// TIA Portal V19 export
DATA_BLOCK "A02_Config"   // DB38
// stored: MemoryReserve 100
   VAR RETAIN
      Area02_Main { ExternalAccessible := 'False'; ExternalVisible := 'False'; ExternalWritable := 'False'} : "AreaConfig";
      RollformingMng : Struct
         SensorsDelayOn : Time := T#100MS;
         SensorsDelayOff : Time := T#500MS;
         SensorExtractor_DelayOn : Time := T#250MS;
         SensorExtractor_DelayOff : Time := T#100MS;
      END_STRUCT;
      PitTableLoop1 : Struct
         LIFT : "ValveMachine_Config";
         Exist : Bool := TRUE;
      END_STRUCT;
      A0201_Profilatrice_RegolazioneFormato : Struct
         Ax_D : Array[1..6] of "Positioning_DOL_Machine_Config";
         Ax_M : Array[7..14] of "Positioning_MOL_Machine_Config";
      END_STRUCT;
      Area02_HU { ExternalAccessible := 'False'; ExternalVisible := 'False'; ExternalWritable := 'False'} : Struct
         Pump { S7_SetPoint := 'True'} : "HU_Pump_Config";
         Tank { S7_SetPoint := 'True'} : "HU_Tank_Config";
      END_STRUCT;
      PostPunchingMatCounter : Struct
         Default_FAK : LReal := 1.0;
      END_STRUCT;
      Rollformer : "PositioningMachine_Config";
      RollfomerLubr { S7_SetPoint := 'True'} : "LubrValve_Config";
      MwFakCalc : Struct
         PushAx : "SpeedMachine_Config";
         Gripper : "ValveMachine_Config";
         MaterialPresenceDly : Time := T#250MS;
         MaterialAbsenceDly : Time := T#250MS;
         PushAx_FwdTimeout { ExternalAccessible := 'False'; ExternalVisible := 'False'; ExternalWritable := 'False'} : Time := T#30S;
         PushAx_BwdTimeout { ExternalAccessible := 'False'; ExternalVisible := 'False'; ExternalWritable := 'False'} : Time := T#30S;
         Default_FAK : LReal := 1.0;
      END_STRUCT;
      FlyingCarriage : "udt_FlyingCarriage_Config";
      FinalCut : Struct
         CheckRestPosition : Bool := TRUE;
         CutHead : "ValveMachine_Config";
         DrawHead : "ValveMachine_Config";
         MarkHead : "ValveMachine_Config";
         Locking : "ValveMachine_Config";
         Locking_AI_HighLimit : Real := 250.0;
         Locking_AI_LowLimit : Real := 0.0;
      END_STRUCT;
      FinalCutLub : Struct
         EnableWngSystemOff : Bool := FALSE;
         ExternalPump : Bool := FALSE;
         PumpWorkDuration : Time := T#2S;
         PumpPauseDuration : Time := T#3S;
         LowTankLevelDly : Time := T#3S;
      END_STRUCT;
      AccRollConveyor : Struct
         Roll1 : "SpeedMachine_Config";
         Roll2 : "SpeedMachine_Config";
         Roll3 : "SpeedMachine_Config";
         PusherVert : Array[1..6] of "ValveMachine_Config";
         PusherHoriz : Array[1..6] of "ValveMachine_Config";
         SensorsDelayOn : Time := T#10MS;
         SensorsDelayOff : Time := T#10MS;
         ExitLeftDelayOn : Time := T#250MS;
         ExitLeftDelayOff : Time := T#250MS;
      END_STRUCT;
   END_VAR
BEGIN
   Area02_Main.TimeOutStopImmediate := T#2S;
   Area02_Main.TimeOutStopInPhase := T#30S;
   Area02_Main.TimeOutStopProgrammed := T#1M;
   Area02_Main.TimeOutResetAlarms := T#1S;
   PitTableLoop1.LIFT.DelayPressureRunningTimeout := T#3S;
   PitTableLoop1.LIFT.DelayMissingCondition := T#3S;
   PitTableLoop1.LIFT.Rest_LsQty := 1;
   PitTableLoop1.LIFT.Work_LsQty := 1;
   PitTableLoop1.LIFT.Rest_RetainAut := FALSE;
   PitTableLoop1.LIFT.Work_RetainAut := FALSE;
   PitTableLoop1.LIFT.V.RestLimSwitchExist := TRUE;
   PitTableLoop1.LIFT.V.WorkLimSwitchExist := TRUE;
   PitTableLoop1.LIFT.V.CheckOilInPressure := FALSE;
   PitTableLoop1.LIFT.V.CutRestWhenIsAtRest := FALSE;
   PitTableLoop1.LIFT.V.CutWorkWhenIsAtWork := FALSE;
   PitTableLoop1.LIFT.V.RestTime := T#1MS;
   PitTableLoop1.LIFT.V.WorkTime := T#1MS;
   PitTableLoop1.LIFT.V.RestTimeOut := T#10S;
   PitTableLoop1.LIFT.V.WorkTimeOut := T#10S;
   A0201_Profilatrice_RegolazioneFormato.Ax_D[1..6].DelayMissingCondition := T#3S;
   A0201_Profilatrice_RegolazioneFormato.Ax_D[1..6].CyclicOBTime_ms := 10.0;
   A0201_Profilatrice_RegolazioneFormato.Ax_D[1..6].Ax.limitMinus := 0.0;
   A0201_Profilatrice_RegolazioneFormato.Ax_D[1..6].Ax.limitPlus := 0.0;
   A0201_Profilatrice_RegolazioneFormato.Ax_D[1..6].Ax.Backlash := 0.4;
   A0201_Profilatrice_RegolazioneFormato.Ax_D[1..6].Ax.BacklashActivation := TRUE;
   A0201_Profilatrice_RegolazioneFormato.Ax_D[1..6].Ax.ToleranceWindow := 0.0;
   A0201_Profilatrice_RegolazioneFormato.Ax_D[1..6].Ax.ToleranceWindowDelay := T#100MS;
   A0201_Profilatrice_RegolazioneFormato.Ax_D[1..6].Ax.PreCutOff := 0.0;
   A0201_Profilatrice_RegolazioneFormato.Ax_D[1..6].Ax.PreEndLowSpeed := 0.0;
   A0201_Profilatrice_RegolazioneFormato.Ax_D[1..6].Ax.PreEndMedSpeed := 0.0;
   A0201_Profilatrice_RegolazioneFormato.Ax_D[1..6].Ax.ChangeDirectionDelay := T#0MS;
   A0201_Profilatrice_RegolazioneFormato.Ax_D[1..6].Ax.StandstillVelocity := 0.5;
   A0201_Profilatrice_RegolazioneFormato.Ax_D[1..6].Ax.StandStillDelay := T#100MS;
   A0201_Profilatrice_RegolazioneFormato.Ax_D[1..6].Ax.HomingDirection := FALSE;
   A0201_Profilatrice_RegolazioneFormato.Ax_D[1..6].Ax.RecallTime := 0.0;
   A0201_Profilatrice_RegolazioneFormato.Ax_D[1..6].Ax.VelocityFilter_T := 10.0;
   A0201_Profilatrice_RegolazioneFormato.Ax_D[1..6].Ax.VelocityMeasUnit := 2;
   A0201_Profilatrice_RegolazioneFormato.Ax_D[1..6].Ax.PosFbkDisabled := FALSE;
   A0201_Profilatrice_RegolazioneFormato.Ax_D[1..6].Ax.FbkCtrlDisabled := TRUE;
   A0201_Profilatrice_RegolazioneFormato.Ax_D[1..6].Ax_UM2."m" := -1.0;
   A0201_Profilatrice_RegolazioneFormato.Ax_D[1].Ax_UM2.q := 267.4;
   A0201_Profilatrice_RegolazioneFormato.Ax_D[2].Ax_UM2.q := 267.3;
   A0201_Profilatrice_RegolazioneFormato.Ax_D[3].Ax_UM2.q := 262.3;
   A0201_Profilatrice_RegolazioneFormato.Ax_D[4].Ax_UM2.q := 262.6;
   A0201_Profilatrice_RegolazioneFormato.Ax_D[5].Ax_UM2.q := 261.8;
   A0201_Profilatrice_RegolazioneFormato.Ax_D[6].Ax_UM2.q := 262.0;
   A0201_Profilatrice_RegolazioneFormato.Ax_D[1..6].S120.SpeedMotor.ReferenceVelocity := 2200.0;
   A0201_Profilatrice_RegolazioneFormato.Ax_D[1..6].S120.SpeedMotor.InvertDirection := FALSE;
   A0201_Profilatrice_RegolazioneFormato.Ax_D[1..6].S120.PowerOffDelay := T#1S_500MS;
   A0201_Profilatrice_RegolazioneFormato.Ax_D[1..6].S120.StandstillVelocity := 20.0;
   A0201_Profilatrice_RegolazioneFormato.Ax_D[1..6].S120.AccTime := 0.5;
   A0201_Profilatrice_RegolazioneFormato.Ax_D[1..6].S120.DecTime := 0.5;
   A0201_Profilatrice_RegolazioneFormato.Ax_D[1..6].Fan.Presence := FALSE;
   A0201_Profilatrice_RegolazioneFormato.Ax_D[1..6].Fan.DelayOff := T#10M;
   A0201_Profilatrice_RegolazioneFormato.Ax_D[1..6].Brake_Presence := FALSE;
   A0201_Profilatrice_RegolazioneFormato.Ax_M[7..14].DelayMissingCondition := T#0MS;
   A0201_Profilatrice_RegolazioneFormato.Ax_M[7..14].CyclicOBTime_ms := 10.0;
   A0201_Profilatrice_RegolazioneFormato.Ax_M[7..14].Ax.limitMinus := 0.0;
   A0201_Profilatrice_RegolazioneFormato.Ax_M[7..14].Ax.limitPlus := 0.0;
   A0201_Profilatrice_RegolazioneFormato.Ax_M[7..14].Ax.Backlash := 0.4;
   A0201_Profilatrice_RegolazioneFormato.Ax_M[7..14].Ax.BacklashActivation := TRUE;
   A0201_Profilatrice_RegolazioneFormato.Ax_M[7..14].Ax.ToleranceWindow := 0.0;
   A0201_Profilatrice_RegolazioneFormato.Ax_M[7..14].Ax.ToleranceWindowDelay := T#100MS;
   A0201_Profilatrice_RegolazioneFormato.Ax_M[7..14].Ax.PreCutOff := 0.0;
   A0201_Profilatrice_RegolazioneFormato.Ax_M[7..14].Ax.PreEndLowSpeed := 0.0;
   A0201_Profilatrice_RegolazioneFormato.Ax_M[7..14].Ax.PreEndMedSpeed := 0.0;
   A0201_Profilatrice_RegolazioneFormato.Ax_M[7..14].Ax.ChangeDirectionDelay := T#0MS;
   A0201_Profilatrice_RegolazioneFormato.Ax_M[7..14].Ax.StandstillVelocity := 0.5;
   A0201_Profilatrice_RegolazioneFormato.Ax_M[7..14].Ax.StandStillDelay := T#100MS;
   A0201_Profilatrice_RegolazioneFormato.Ax_M[7..14].Ax.HomingDirection := FALSE;
   A0201_Profilatrice_RegolazioneFormato.Ax_M[7..14].Ax.RecallTime := 0.0;
   A0201_Profilatrice_RegolazioneFormato.Ax_M[7..14].Ax.VelocityFilter_T := 10.0;
   A0201_Profilatrice_RegolazioneFormato.Ax_M[7..14].Ax.VelocityMeasUnit := 2;
   A0201_Profilatrice_RegolazioneFormato.Ax_M[7..14].Ax.PosFbkDisabled := FALSE;
   A0201_Profilatrice_RegolazioneFormato.Ax_M[7..14].Ax.FbkCtrlDisabled := TRUE;
   A0201_Profilatrice_RegolazioneFormato.Ax_M[7..8].Ax_UM2."m" := -1.0;
   A0201_Profilatrice_RegolazioneFormato.Ax_M[9..10].Ax_UM2."m" := 1.0;
   A0201_Profilatrice_RegolazioneFormato.Ax_M[11..14].Ax_UM2."m" := -1.0;
   A0201_Profilatrice_RegolazioneFormato.Ax_M[7..8].Ax_UM2.q := 84.8;
   A0201_Profilatrice_RegolazioneFormato.Ax_M[9..10].Ax_UM2.q := 0.0;
   A0201_Profilatrice_RegolazioneFormato.Ax_M[11..12].Ax_UM2.q := 81.6;
   A0201_Profilatrice_RegolazioneFormato.Ax_M[13..14].Ax_UM2.q := 81.3;
   Area02_HU.Pump.SafetyCutOffValveExist := TRUE;
   Area02_HU.Pump.StandbyValveExist := TRUE;
   Area02_HU.Pump.OilPumpContactotFeedbackTimeOut := T#5S;
   Area02_HU.Tank.RecirculationPumpExist := TRUE;
   Area02_HU.Tank.HeatExchangerFanExist := TRUE;
   Area02_HU.Tank.HeatingUnitExistNum := 1;
   Area02_HU.Tank.ChillerExist := FALSE;
   Area02_HU.Tank.OilMaxTemperature := 70.0;
   Area02_HU.Tank.WaterMaxTemperature := 60.0;
   Area02_HU.Tank.TemperatureStartCheckFilters := 35.0;
   Area02_HU.Tank.HeatingHysteresys := 1.0;
   Area02_HU.Tank.DelayHeatingStart := T#30S;
   Area02_HU.Tank.DelayHeatingStop := T#30S;
   Area02_HU.Tank.DelayCollingStart := T#30S;
   Area02_HU.Tank.DelayCollingStop := T#30S;
   Area02_HU.Tank.AnlOilTemp_HighLimit := 100.0;
   Area02_HU.Tank.AnlOilTemp_LowLimit := 0.0;
   Area02_HU.Tank.AnlWaterTemp_HighLimit := 100.0;
   Area02_HU.Tank.AnlWaterTemp_LowLimit := -10.0;
   Rollformer.SLS_VEL := 5000.0;
   Rollformer.DelayMissingCondition := T#3S;
   Rollformer.Ax.OptionON_EncoderSelection := FALSE;
   Rollformer.Ax.OptionON_ParameterChange := TRUE;
   Rollformer.Ax.OptionON_AutoReloadPosition := TRUE;
   Rollformer.Ax.OptionON_ManPreset := FALSE;
   Rollformer.Ax.HomeMode := 0;
   Rollformer.Ax.PosAxis.Simulation := FALSE;
   Rollformer.Ax.PosAxis.PowerOffDelay := T#5S;
   Rollformer.Ax.PosAxis.PowerStartMode := 1;
   Rollformer.Ax.PosAxis.PowerStopMode := 2;
   Rollformer.Fan.Presence := TRUE;
   Rollformer.Fan.DelayOff := T#10M;
   Rollformer.Brake_Presence := FALSE;
   RollfomerLubr.WorkMode := 2;
   RollfomerLubr.CounterMode := 0;
   RollfomerLubr.ValveType := 1;
   RollfomerLubr.ManualCmdTimeOut := T#5M;
   MwFakCalc.PushAx.SLS_VEL := 5000.0;
   MwFakCalc.PushAx.DelayMissingCondition := T#3S;
   MwFakCalc.PushAx.Ax.SINA_Drive.ReferenceVelocity := 2200.0;
   MwFakCalc.PushAx.Ax.SINA_Drive.InvertDirection := FALSE;
   MwFakCalc.PushAx.Ax.MinAccTime := 0.1;
   MwFakCalc.PushAx.Ax.MinDecTime := 0.1;
   MwFakCalc.PushAx.Ax.LeadScrewPitchVal := 79.984948;
   MwFakCalc.PushAx.Ax.MotorRevolution := 5.0;
   MwFakCalc.PushAx.Ax.LoadRevolution := 1.0;
   MwFakCalc.PushAx.Ax.PowerOffDelay := T#1S_500MS;
   MwFakCalc.PushAx.Ax.StandstillVelocity := 20.0;
   MwFakCalc.PushAx.Ax.StandstillDelay := T#100MS;
   MwFakCalc.PushAx.Fan.Presence := FALSE;
   MwFakCalc.PushAx.Fan.DelayOff := T#0MS;
   MwFakCalc.PushAx.Brake_Presence := FALSE;
   MwFakCalc.Gripper.DelayPressureRunningTimeout := T#3S;
   MwFakCalc.Gripper.DelayMissingCondition := T#3S;
   MwFakCalc.Gripper.Rest_LsQty := 1;
   MwFakCalc.Gripper.Work_LsQty := 1;
   MwFakCalc.Gripper.Rest_RetainAut := FALSE;
   MwFakCalc.Gripper.Work_RetainAut := FALSE;
   MwFakCalc.Gripper.V.RestLimSwitchExist := TRUE;
   MwFakCalc.Gripper.V.WorkLimSwitchExist := TRUE;
   MwFakCalc.Gripper.V.CheckOilInPressure := FALSE;
   MwFakCalc.Gripper.V.CutRestWhenIsAtRest := TRUE;
   MwFakCalc.Gripper.V.CutWorkWhenIsAtWork := TRUE;
   MwFakCalc.Gripper.V.RestTime := T#1MS;
   MwFakCalc.Gripper.V.WorkTime := T#1MS;
   MwFakCalc.Gripper.V.RestTimeOut := T#1S;
   MwFakCalc.Gripper.V.WorkTimeOut := T#1S;
   FlyingCarriage.SLS_VEL := 5000.0;
   FlyingCarriage.DelayMissingCondition := T#3S;
   FlyingCarriage.Fan.Exist := FALSE;
   FlyingCarriage.Fan.DelayOff := T#15M;
   FinalCut.CutHead.DelayPressureRunningTimeout := T#3S;
   FinalCut.CutHead.DelayMissingCondition := T#3S;
   FinalCut.CutHead.Rest_LsQty := 1;
   FinalCut.CutHead.Work_LsQty := 1;
   FinalCut.CutHead.Rest_RetainAut := FALSE;
   FinalCut.CutHead.Work_RetainAut := FALSE;
   FinalCut.CutHead.V.RestLimSwitchExist := TRUE;
   FinalCut.CutHead.V.WorkLimSwitchExist := TRUE;
   FinalCut.CutHead.V.CheckOilInPressure := TRUE;
   FinalCut.CutHead.V.CutRestWhenIsAtRest := FALSE;
   FinalCut.CutHead.V.CutWorkWhenIsAtWork := FALSE;
   FinalCut.CutHead.V.RestTime := T#1MS;
   FinalCut.CutHead.V.WorkTime := T#1MS;
   FinalCut.CutHead.V.RestTimeOut := T#1S_500MS;
   FinalCut.CutHead.V.WorkTimeOut := T#1S_500MS;
   FinalCut.DrawHead.DelayPressureRunningTimeout := T#3S;
   FinalCut.DrawHead.DelayMissingCondition := T#3S;
   FinalCut.DrawHead.Rest_LsQty := 1;
   FinalCut.DrawHead.Work_LsQty := 1;
   FinalCut.DrawHead.Rest_RetainAut := FALSE;
   FinalCut.DrawHead.Work_RetainAut := FALSE;
   FinalCut.DrawHead.V.RestLimSwitchExist := TRUE;
   FinalCut.DrawHead.V.WorkLimSwitchExist := TRUE;
   FinalCut.DrawHead.V.CheckOilInPressure := TRUE;
   FinalCut.DrawHead.V.CutRestWhenIsAtRest := FALSE;
   FinalCut.DrawHead.V.CutWorkWhenIsAtWork := FALSE;
   FinalCut.DrawHead.V.RestTime := T#1MS;
   FinalCut.DrawHead.V.WorkTime := T#1MS;
   FinalCut.DrawHead.V.RestTimeOut := T#1S_500MS;
   FinalCut.DrawHead.V.WorkTimeOut := T#1S_500MS;
   FinalCut.MarkHead.DelayPressureRunningTimeout := T#3S;
   FinalCut.MarkHead.DelayMissingCondition := T#3S;
   FinalCut.MarkHead.Rest_LsQty := 1;
   FinalCut.MarkHead.Work_LsQty := 1;
   FinalCut.MarkHead.Rest_RetainAut := FALSE;
   FinalCut.MarkHead.Work_RetainAut := FALSE;
   FinalCut.MarkHead.V.RestLimSwitchExist := TRUE;
   FinalCut.MarkHead.V.WorkLimSwitchExist := TRUE;
   FinalCut.MarkHead.V.CheckOilInPressure := TRUE;
   FinalCut.MarkHead.V.CutRestWhenIsAtRest := FALSE;
   FinalCut.MarkHead.V.CutWorkWhenIsAtWork := FALSE;
   FinalCut.MarkHead.V.RestTime := T#1MS;
   FinalCut.MarkHead.V.WorkTime := T#1MS;
   FinalCut.MarkHead.V.RestTimeOut := T#1S_500MS;
   FinalCut.MarkHead.V.WorkTimeOut := T#1S_500MS;
   FinalCut.Locking.DelayPressureRunningTimeout := T#3S;
   FinalCut.Locking.DelayMissingCondition := T#3S;
   FinalCut.Locking.Rest_LsQty := 1;
   FinalCut.Locking.Work_LsQty := 1;
   FinalCut.Locking.Rest_RetainAut := FALSE;
   FinalCut.Locking.Work_RetainAut := FALSE;
   FinalCut.Locking.V.RestLimSwitchExist := TRUE;
   FinalCut.Locking.V.WorkLimSwitchExist := TRUE;
   FinalCut.Locking.V.CheckOilInPressure := TRUE;
   FinalCut.Locking.V.CutRestWhenIsAtRest := FALSE;
   FinalCut.Locking.V.CutWorkWhenIsAtWork := FALSE;
   FinalCut.Locking.V.RestTime := T#1MS;
   FinalCut.Locking.V.WorkTime := T#1MS;
   FinalCut.Locking.V.RestTimeOut := T#2S;
   FinalCut.Locking.V.WorkTimeOut := T#2S;
   AccRollConveyor.Roll1.SLS_VEL := 5000.0;
   AccRollConveyor.Roll1.DelayMissingCondition := T#3S;
   AccRollConveyor.Roll1.Ax.SINA_Drive.ReferenceVelocity := 2200.0;
   AccRollConveyor.Roll1.Ax.SINA_Drive.InvertDirection := FALSE;
   AccRollConveyor.Roll1.Ax.MinAccTime := 0.1;
   AccRollConveyor.Roll1.Ax.MinDecTime := 0.1;
   AccRollConveyor.Roll1.Ax.LeadScrewPitchVal := 219.911;
   AccRollConveyor.Roll1.Ax.MotorRevolution := 7.0;
   AccRollConveyor.Roll1.Ax.LoadRevolution := 1.0;
   AccRollConveyor.Roll1.Ax.PowerOffDelay := T#1S_500MS;
   AccRollConveyor.Roll1.Ax.StandstillVelocity := 50.0;
   AccRollConveyor.Roll1.Ax.StandstillDelay := T#100MS;
   AccRollConveyor.Roll1.Fan.Presence := FALSE;
   AccRollConveyor.Roll1.Fan.DelayOff := T#0MS;
   AccRollConveyor.Roll1.Brake_Presence := FALSE;
   AccRollConveyor.Roll2.SLS_VEL := 5000.0;
   AccRollConveyor.Roll2.DelayMissingCondition := T#3S;
   AccRollConveyor.Roll2.Ax.SINA_Drive.ReferenceVelocity := 2200.0;
   AccRollConveyor.Roll2.Ax.SINA_Drive.InvertDirection := FALSE;
   AccRollConveyor.Roll2.Ax.MinAccTime := 0.1;
   AccRollConveyor.Roll2.Ax.MinDecTime := 0.1;
   AccRollConveyor.Roll2.Ax.LeadScrewPitchVal := 219.911;
   AccRollConveyor.Roll2.Ax.MotorRevolution := 7.0;
   AccRollConveyor.Roll2.Ax.LoadRevolution := 1.0;
   AccRollConveyor.Roll2.Ax.PowerOffDelay := T#1S_500MS;
   AccRollConveyor.Roll2.Ax.StandstillVelocity := 50.0;
   AccRollConveyor.Roll2.Ax.StandstillDelay := T#100MS;
   AccRollConveyor.Roll2.Fan.Presence := FALSE;
   AccRollConveyor.Roll2.Fan.DelayOff := T#0MS;
   AccRollConveyor.Roll2.Brake_Presence := FALSE;
   AccRollConveyor.Roll3.SLS_VEL := 5000.0;
   AccRollConveyor.Roll3.DelayMissingCondition := T#3S;
   AccRollConveyor.Roll3.Ax.SINA_Drive.ReferenceVelocity := 2200.0;
   AccRollConveyor.Roll3.Ax.SINA_Drive.InvertDirection := FALSE;
   AccRollConveyor.Roll3.Ax.MinAccTime := 0.1;
   AccRollConveyor.Roll3.Ax.MinDecTime := 0.1;
   AccRollConveyor.Roll3.Ax.LeadScrewPitchVal := 219.911;
   AccRollConveyor.Roll3.Ax.MotorRevolution := 7.0;
   AccRollConveyor.Roll3.Ax.LoadRevolution := 1.0;
   AccRollConveyor.Roll3.Ax.PowerOffDelay := T#1S_500MS;
   AccRollConveyor.Roll3.Ax.StandstillVelocity := 50.0;
   AccRollConveyor.Roll3.Ax.StandstillDelay := T#100MS;
   AccRollConveyor.Roll3.Fan.Presence := FALSE;
   AccRollConveyor.Roll3.Fan.DelayOff := T#0MS;
   AccRollConveyor.Roll3.Brake_Presence := FALSE;
   AccRollConveyor.PusherVert[1..6].DelayPressureRunningTimeout := T#3S;
   AccRollConveyor.PusherVert[1..6].DelayMissingCondition := T#3S;
   AccRollConveyor.PusherVert[1..6].Rest_LsQty := 1;
   AccRollConveyor.PusherVert[1..6].Work_LsQty := 1;
   AccRollConveyor.PusherVert[1..6].Rest_RetainAut := FALSE;
   AccRollConveyor.PusherVert[1..6].Work_RetainAut := FALSE;
   AccRollConveyor.PusherVert[1..6].V.RestLimSwitchExist := TRUE;
   AccRollConveyor.PusherVert[1..6].V.WorkLimSwitchExist := FALSE;
   AccRollConveyor.PusherVert[1..6].V.CheckOilInPressure := FALSE;
   AccRollConveyor.PusherVert[1..6].V.CutRestWhenIsAtRest := FALSE;
   AccRollConveyor.PusherVert[1..6].V.CutWorkWhenIsAtWork := FALSE;
   AccRollConveyor.PusherVert[1..6].V.RestTime := T#1MS;
   AccRollConveyor.PusherVert[1..6].V.WorkTime := T#250MS;
   AccRollConveyor.PusherVert[1..6].V.RestTimeOut := T#1S_500MS;
   AccRollConveyor.PusherVert[1..6].V.WorkTimeOut := T#1S_500MS;
   AccRollConveyor.PusherHoriz[1..6].DelayPressureRunningTimeout := T#3S;
   AccRollConveyor.PusherHoriz[1..6].DelayMissingCondition := T#3S;
   AccRollConveyor.PusherHoriz[1..6].Rest_LsQty := 1;
   AccRollConveyor.PusherHoriz[1..6].Work_LsQty := 1;
   AccRollConveyor.PusherHoriz[1..6].Rest_RetainAut := FALSE;
   AccRollConveyor.PusherHoriz[1..6].Work_RetainAut := FALSE;
   AccRollConveyor.PusherHoriz[1..6].V.RestLimSwitchExist := TRUE;
   AccRollConveyor.PusherHoriz[1..6].V.WorkLimSwitchExist := TRUE;
   AccRollConveyor.PusherHoriz[1..6].V.CheckOilInPressure := FALSE;
   AccRollConveyor.PusherHoriz[1..6].V.CutRestWhenIsAtRest := FALSE;
   AccRollConveyor.PusherHoriz[1..6].V.CutWorkWhenIsAtWork := FALSE;
   AccRollConveyor.PusherHoriz[1..6].V.RestTime := T#1MS;
   AccRollConveyor.PusherHoriz[1..6].V.WorkTime := T#1MS;
   AccRollConveyor.PusherHoriz[1..6].V.RestTimeOut := T#1S_500MS;
   AccRollConveyor.PusherHoriz[1..6].V.WorkTimeOut := T#1S_500MS;
END_DATA_BLOCK
